// Mitsubishi GX Works2 project: Group4_V9   PLC: FX3G

// global labels: Global1
VAR_GLOBAL
  On_Switch AT X007 : BOOL;
END_VAR
VAR_GLOBAL CONSTANT
  Min_Cream : REAL := 300;
  Min_Biscuit : REAL := 6;
  Min_Choc : REAL := 120;
END_VAR
VAR_GLOBAL
  light AT Y007 : BOOL;
  Piping_Start AT X011 : BOOL;
  Whipped_Cream_Piping AT D2100 : REAL;
  Start_System AT X010 : BOOL;
  System_On AT M0 : BOOL;
  Malfunction_Status AT X005 : BOOL;
  Sen_Touch AT X001 : BOOL;
  Sen_Camera AT X002 : BOOL;
  Sen_30 AT X003 : BOOL;
  Machine AT Y004 : BOOL;
  Sen_15 AT X004 : BOOL;
  Biscuit_tray AT D2300 : REAL;
  ziluf AT M2 : BOOL;
  Blink AT M1 : BOOL;
  Blink1 AT Y000 : BOOL;
  TS_1 AT TS1 : BOOL;
  TS_2 AT TS2 : BOOL;
  Blink2 AT Y001 : BOOL;
  Check_Inv AT M17 : BOOL;
  Start_Day AT M1 : BOOL;
  Biscuit_Input AT D1333 : REAL;
  Chocolate_Input AT D1222 : REAL;
  Whipped_Cream_Input AT D1111 : REAL;
  Biscuit_Inv AT D1300 : REAL;
  Chocolate_Inv AT D1200 : REAL;
  Whipped_Cream_Inv AT D1100 : REAL;
  Full_Inv AT M107 : BOOL;
  Factory_working AT M117 : BOOL;
  Biscuit_Suff AT M130 : BOOL;
  Chocolate_Suff AT M120 : BOOL;
  Cream_Suff AT M110 : BOOL;
  Start_Glaze AT X006 : BOOL;
END_VAR
VAR_GLOBAL CONSTANT
  Double_Layer : INT := 6;
  Single_Layer : REAL := 5;
END_VAR
VAR_GLOBAL
  analog_Input_1 AT D8280 : INT;
  Single_Layer_Only AT M30 : BOOL;
END_VAR
VAR_GLOBAL CONSTANT
  Double_Layer_Amount : REAL := 240;
  Single_Layer_Amount : REAL := 120;
END_VAR
VAR_GLOBAL
  Chocolate_Dipping AT D2200 : REAL;
  Dipping_Time AT TC5 : BOOL;
  Dipping_Timer AT TC5 : BOOL;
  Dipping_Light AT Y003 : BOOL;
END_VAR
VAR_GLOBAL CONSTANT
  Double_Layer_Min : REAL := 6;
  Double_Layer_Max : REAL := 10;
  normalization : REAL := 390;
END_VAR
VAR_GLOBAL
  AnalogInput AT M33 : BOOL;
  Dip_Option AT D2220 : REAL;
  DSSD AT Y002 : BOOL;
  End_Packing AT Y002 : BOOL;
  TCoil0 AT TC0 : BOOL;
  MachineB AT D2400 : REAL;
  M_11 AT M11 : BOOL;
  TCoil1 AT TC1 : BOOL;
  M_7 AT M7 : BOOL;
  TCoil2 AT TC2 : BOOL;
  Dipping_Done AT M333 : BOOL;
  Packing_Creambo AT X000 : BOOL;
  Creambo_Counter AT CC1 : BOOL;
END_VAR
VAR_GLOBAL CONSTANT
  Creambo_5 : INT := 5;
END_VAR
VAR_GLOBAL
  Creambo_Counter_On AT CS1 : BOOL;
  last_Creambo_Warning AT Y002 : BOOL;
  Done_Packing_Counter AT CC2 : BOOL;
END_VAR
VAR_GLOBAL CONSTANT
  All_Creambo_packed : INT := 6;
END_VAR
VAR_GLOBAL
  Creambo_Done_counter AT CS2 : BOOL;
  Finished_Creambos_Sum AT D6666 : REAL;
END_VAR
VAR_GLOBAL CONSTANT
  Packed_Creambo_sixpack : REAL := 6;
END_VAR
VAR_GLOBAL
  Finished_Iteration AT M238 : BOOL;
  TC_7 AT TC7 : BOOL;
  TS_90 AT TS90 : BOOL;
  M_20 AT M20 : BOOL;
  Piping_Finished AT M200 : BOOL;
  Reset_Iteration AT M2000 : BOOL;
  Start_Glaze_Ready AT M106 : BOOL;
  Choc_Inv AT M120 : BOOL;
  Turn_Off_Inv_Check AT M227 : BOOL;
  Turn_Off_Help_Lights AT M227 : BOOL;
  TCoil3 AT TC3 : BOOL;
  TS_3 AT TS3 : BOOL;
  light_flick AT M52 : BOOL;
  TS_0 AT TS0 : BOOL;
  analog_output AT D8282 : INT;
  M_6 AT M6 : BOOL;
  M_8 AT M8 : BOOL;
END_VAR
VAR_GLOBAL CONSTANT
  normalization_back : REAL := 40;
END_VAR
VAR_GLOBAL
  M_98 AT M98 : BOOL;
  M_88 AT M88 : BOOL;
  TS_67 AT TS67 : BOOL;
  TCoil4 AT TC4 : BOOL;
  TS_4 AT TS4 : BOOL;
  M_56 AT M56 : BOOL;
  last_Iteration AT M255 : BOOL;
  Creambo_Normalized AT D6060 : REAL;
END_VAR

// task Task_01 (event TRUE, interval 0, priority 31): POU_01

PROGRAM POU_01
VAR CONSTANT
  M_10 : BOOL;
END_VAR
(* structured ladder/FBD written out as ST: instructions are called as NAME(EN, inputs, outputs); _pN, _eN, _tN stand for wires *)
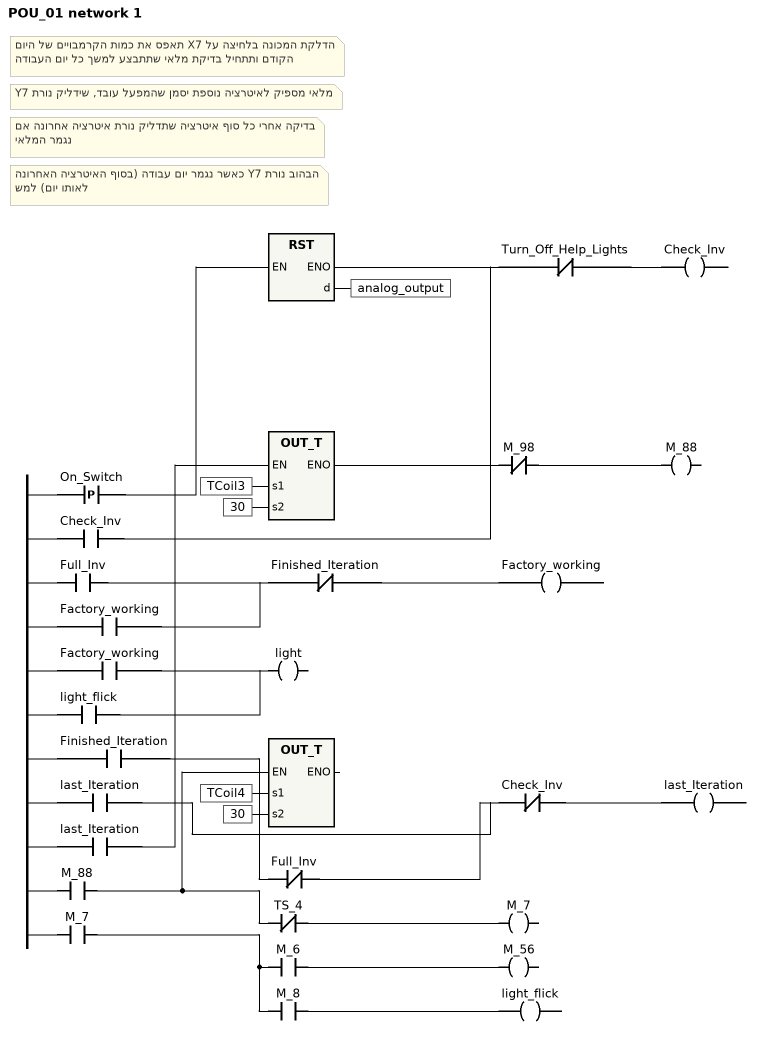
(* network 1 *)
(* הדלקת המכונה בלחיצה על X7 תאפס את כמות הקרמבויים של היום הקודם ותתחיל בדיקת מלאי שתתבצע למשך כל יום העבודה *)
(* מלאי מספיק לאיטרציה נוספת יסמן שהמפעל עובד, שידליק נורת Y7 *)
(* בדיקה אחרי כל סוף איטרציה שתדליק נורת איטרציה אחרונה אם נגמר המלאי *)
(* הבהוב נורת Y7 כאשר נגמר יום עבודה (בסוף האיטרציה האחרונה לאותו יום) למש *)
_e1 := RST(LDP(TRUE, On_Switch), analog_output);
Check_Inv := (_e1 OR Check_Inv) AND NOT Turn_Off_Help_Lights;
Factory_working := (Full_Inv OR Factory_working) AND NOT Finished_Iteration;
light := Factory_working OR light_flick;
last_Iteration := ((Finished_Iteration AND NOT Full_Inv) OR last_Iteration) AND NOT Check_Inv;
_e2 := OUT_T(last_Iteration, TCoil3, 30);
M_88 := _e2 AND NOT M_98;
OUT_T(M_88, TCoil4, 30);
M_7 := M_88 AND NOT TS_4;
M_56 := M_7 AND M_6;
light_flick := M_7 AND M_8;
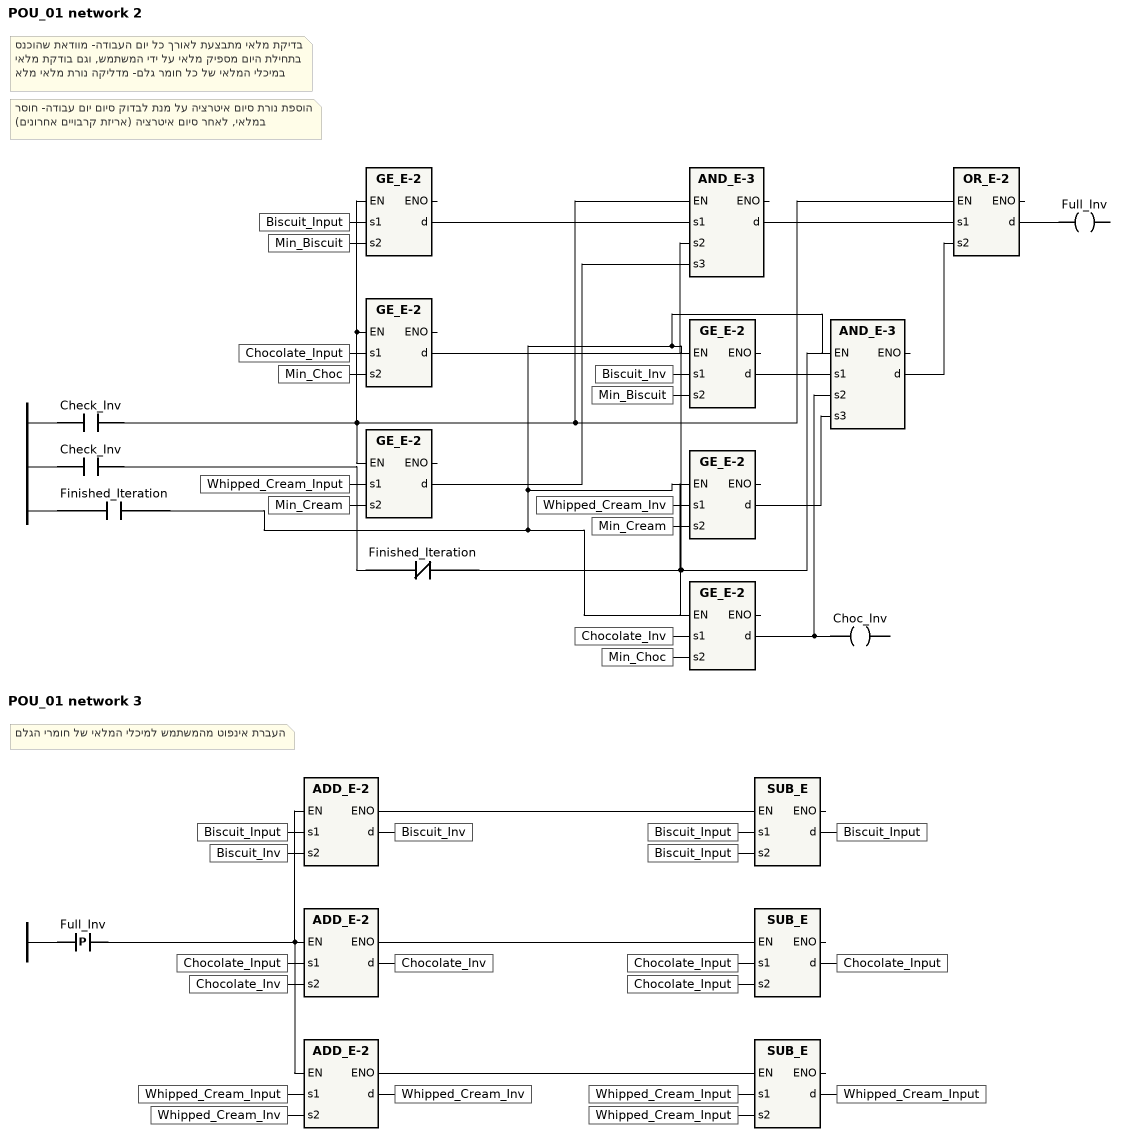
(* network 2 *)
(* בדיקת מלאי מתבצעת לאורך כל יום העבודה- מוודאת שהוכנס בתחילת היום מספיק מלאי על ידי המשתמש, וגם בודקת מלאי במיכלי המלאי של כל חומר גלם- מדליקה נורת מלאי מלא *)
(* הוספת נורת סיום איטרציה על מנת לבדוק סיום יום עבודה- חוסר במלאי, לאחר סיום איטרציה (אריזת קרבויים אחרונים) *)
GE_E(Check_Inv, Biscuit_Input, Min_Biscuit, _t1);
GE_E(Check_Inv, Chocolate_Input, Min_Choc, _t2);
GE_E(Check_Inv, Whipped_Cream_Input, Min_Cream, _t3);
AND_E(Check_Inv, _t1, _t2, _t3, _t4);
_p5 := (Check_Inv AND NOT Finished_Iteration) OR Finished_Iteration;
GE_E(_p5, Biscuit_Inv, Min_Biscuit, _t6);
GE_E(_p5, Chocolate_Inv, Min_Choc, _t7);
GE_E(_p5, Whipped_Cream_Inv, Min_Cream, _t8);
AND_E(_p5, _t6, _t7, _t8, _t9);
OR_E(Check_Inv, _t4, _t9, _t10);
Full_Inv := _t10;
Choc_Inv := _t7;
(* network 3 *)
(* העברת אינפוט מהמשתמש למיכלי המלאי של חומרי הגלם *)
_p1 := LDP(TRUE, Full_Inv);
_e2 := ADD_E(_p1, Biscuit_Input, Biscuit_Inv, Biscuit_Inv);
SUB_E(_e2, Biscuit_Input, Biscuit_Input, Biscuit_Input);
_e3 := ADD_E(_p1, Chocolate_Input, Chocolate_Inv, Chocolate_Inv);
SUB_E(_e3, Chocolate_Input, Chocolate_Input, Chocolate_Input);
_e4 := ADD_E(_p1, Whipped_Cream_Input, Whipped_Cream_Inv, Whipped_Cream_Inv);
SUB_E(_e4, Whipped_Cream_Input, Whipped_Cream_Input, Whipped_Cream_Input);
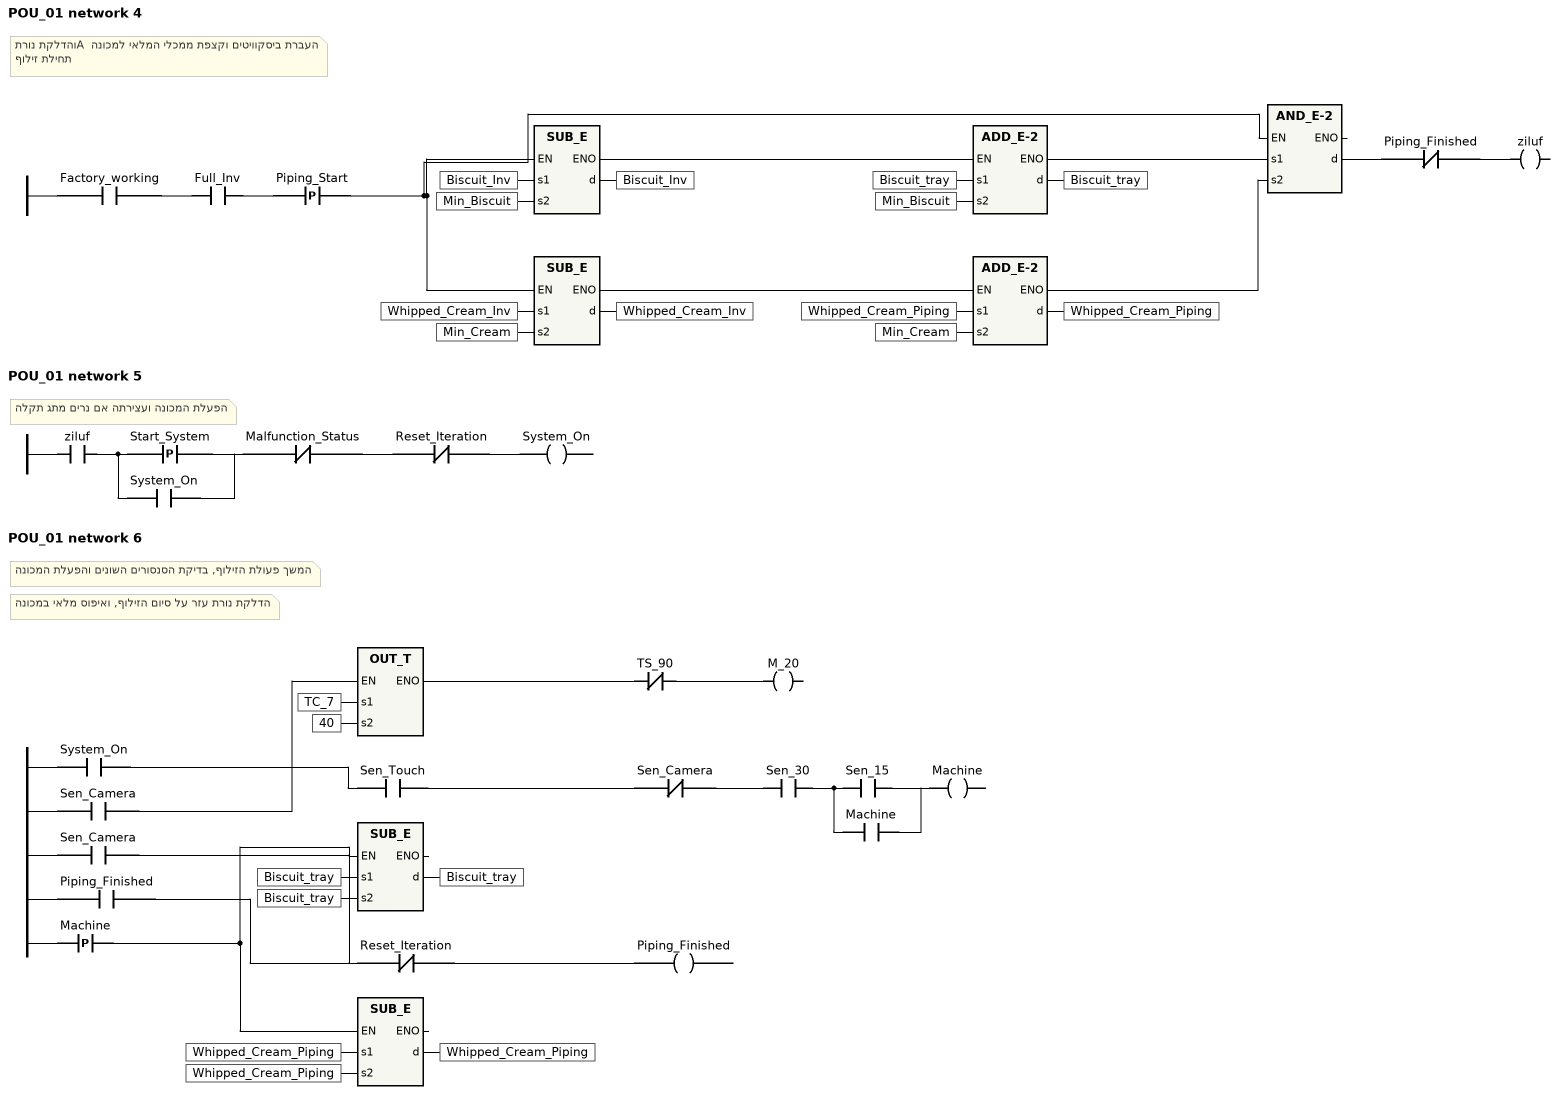
(* network 4 *)
(* העברת ביסקוויטים וקצפת ממכלי המלאי למכונה  Aוהדלקת נורת תחילת זילוף *)
_p1 := Factory_working AND Full_Inv AND LDP(TRUE, Piping_Start);
_e2 := SUB_E(_p1, Biscuit_Inv, Min_Biscuit, Biscuit_Inv);
_e3 := ADD_E(_e2, Biscuit_tray, Min_Biscuit, Biscuit_tray);
_e4 := SUB_E(_p1, Whipped_Cream_Inv, Min_Cream, Whipped_Cream_Inv);
_e5 := ADD_E(_e4, Whipped_Cream_Piping, Min_Cream, Whipped_Cream_Piping);
AND_E(_p1, _e3, _e5, _t6);
ziluf := _t6 AND NOT Piping_Finished;
(* network 5 *)
(* הפעלת המכונה ועצירתה אם נרים מתג תקלה *)
System_On := (((ziluf AND LDP(TRUE, Start_System)) OR (ziluf AND System_On)) AND NOT Malfunction_Status) AND NOT Reset_Iteration;
(* network 6 *)
(* המשך פעולת הזילוף, בדיקת הסנסורים השונים והפעלת המכונה *)
(* הדלקת נורת עזר על סיום הזילוף, ואיפוס מלאי במכונה *)
_p1 := System_On AND Sen_Touch AND NOT Sen_Camera AND Sen_30;
Machine := (_p1 AND Sen_15) OR (_p1 AND Machine);
_e2 := OUT_T(Sen_Camera, TC_7, 40);
M_20 := _e2 AND NOT TS_90;
Piping_Finished := (Sen_Camera OR Piping_Finished) AND NOT Reset_Iteration;
_p3 := LDP(TRUE, Machine);
SUB_E(_p3, Biscuit_tray, Biscuit_tray, Biscuit_tray);
SUB_E(_p3, Whipped_Cream_Piping, Whipped_Cream_Piping, Whipped_Cream_Piping);
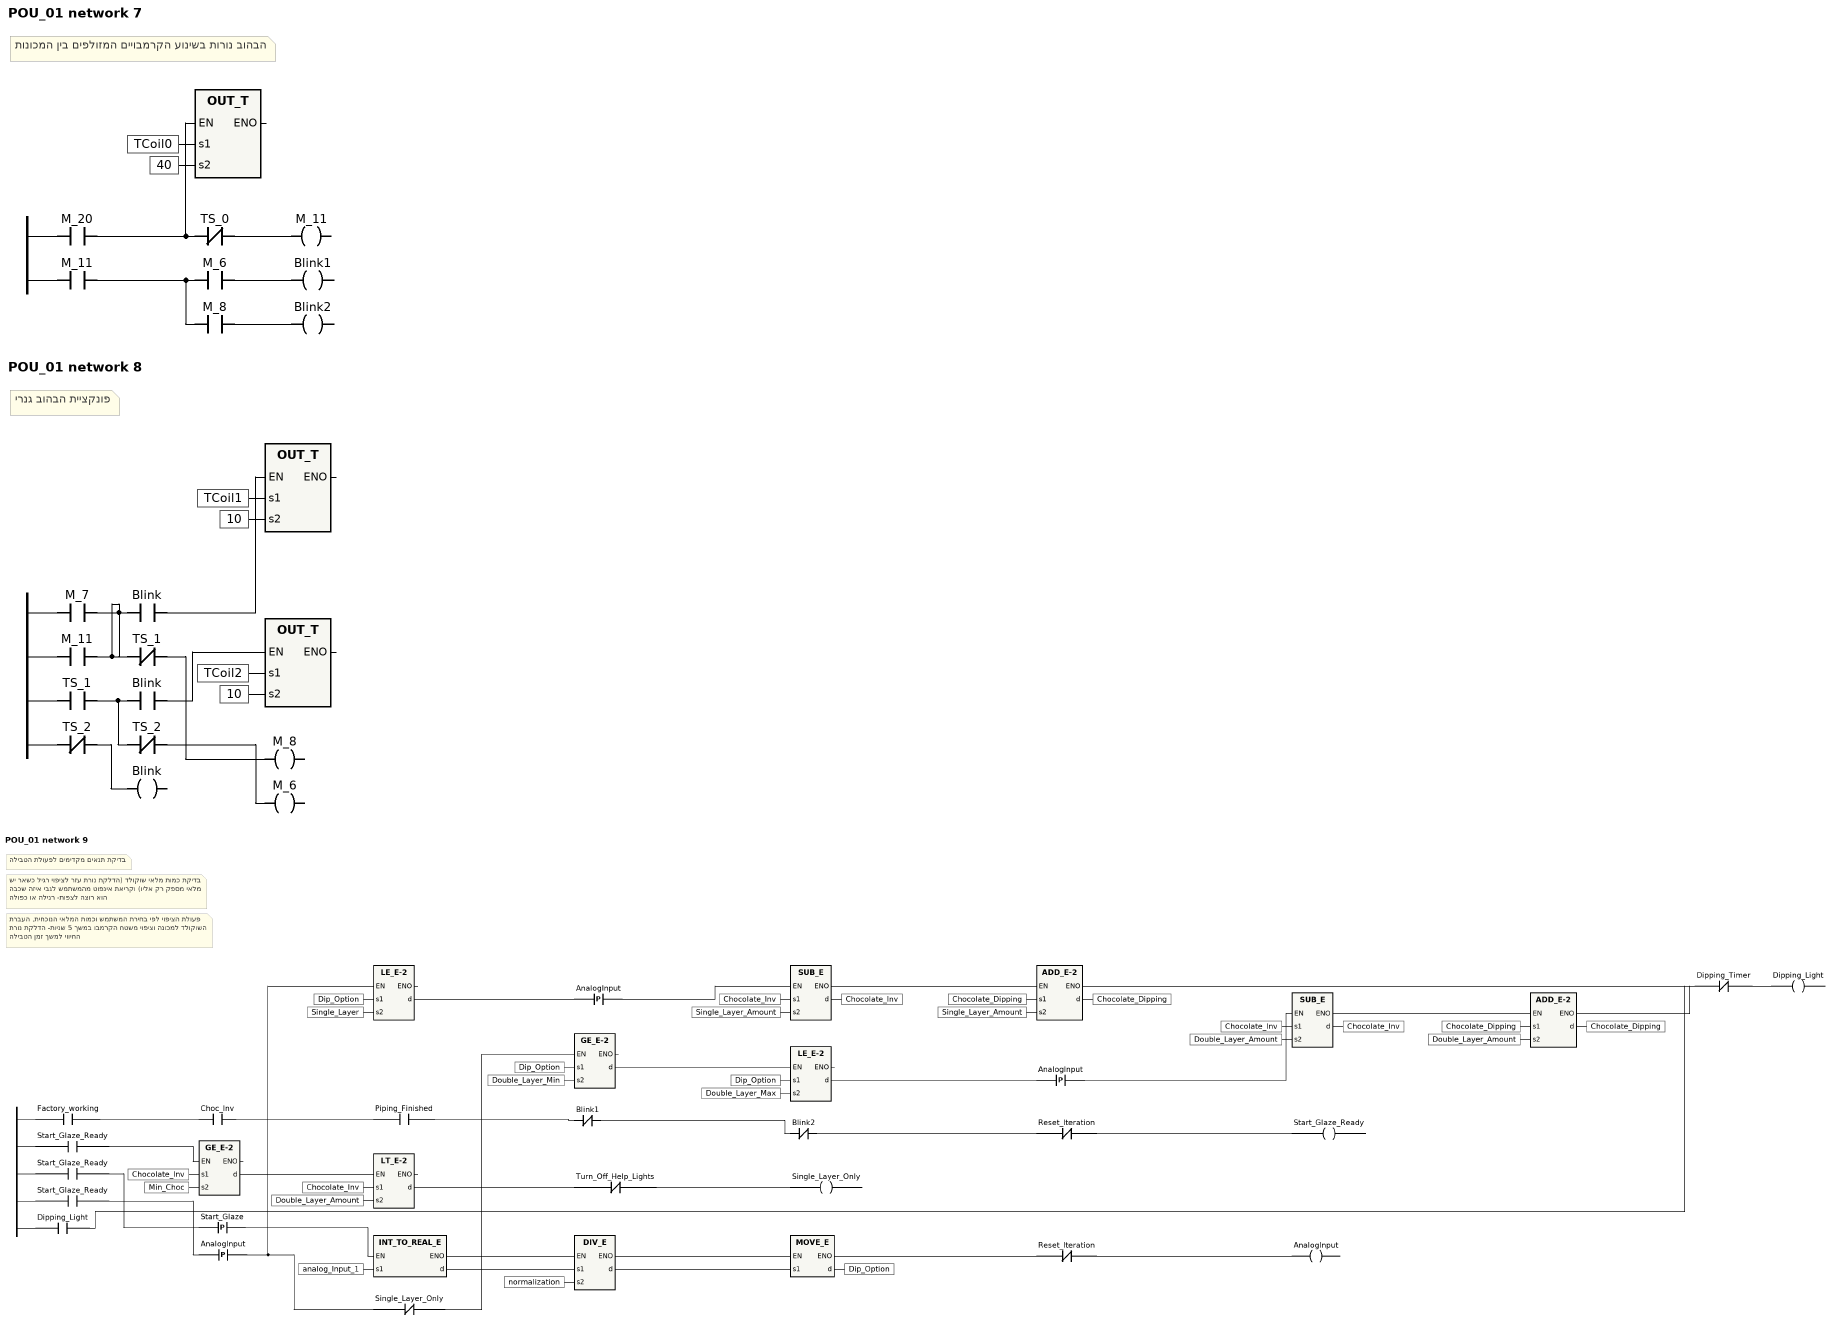
(* network 7 *)
(* הבהוב נורות בשינוע הקרמבויים המזולפים בין המכונות *)
OUT_T(M_20, TCoil0, 40);
M_11 := M_20 AND NOT TS_0;
Blink1 := M_11 AND M_6;
Blink2 := M_11 AND M_8;
(* network 8 *)
(* פונקציית הבהוב גנרי *)
_p1 := M_7 OR M_11;
OUT_T(_p1 AND Blink, TCoil1, 10);
M_8 := _p1 AND NOT TS_1;
OUT_T(TS_1 AND Blink, TCoil2, 10);
M_6 := TS_1 AND NOT TS_2;
Blink := NOT TS_2;
(* network 9 *)
(* בדיקת תנאים מקדימים לפעולת הטבילה *)
(* בדיקת כמות מלאי שוקולד (הדלקת נורת עזר לציפוי רגיל כשאר יש מלאי מספק רק אליו) וקריאת אינפוט מהמשתמש לגבי איזה שכבה הוא רוצה לצפות- רגילה או כפולה *)
(* פעולת הציפוי לפי בחירת המשתמש וכמות המלאי הנוכחית, העברת השוקולד למכונה וציפוי משטח הקרמבו במשך 5 שניות- הדלקת נורת החיווי למשך זמן הטבילה *)
Start_Glaze_Ready := Factory_working AND Choc_Inv AND Piping_Finished AND NOT Blink1 AND NOT Blink2 AND NOT Reset_Iteration;
GE_E(Start_Glaze_Ready, Chocolate_Inv, Min_Choc, _t1);
LT_E(_t1, Chocolate_Inv, Double_Layer_Amount, _t2);
Single_Layer_Only := _t2 AND NOT Turn_Off_Help_Lights;
_e4 := INT_TO_REAL_E(Start_Glaze_Ready AND LDP(TRUE, Start_Glaze), analog_Input_1, _t3);
_e6 := DIV_E(_e4, _t3, normalization, _t5);
_e7 := MOVE_E(_e6, _t5, Dip_Option);
AnalogInput := _e7 AND NOT Reset_Iteration;
_p8 := Start_Glaze_Ready AND LDP(TRUE, AnalogInput);
LE_E(_p8, Dip_Option, Single_Layer, _t9);
_e10 := SUB_E(_t9 AND LDP(TRUE, AnalogInput), Chocolate_Inv, Single_Layer_Amount, Chocolate_Inv);
_e11 := ADD_E(_e10, Chocolate_Dipping, Single_Layer_Amount, Chocolate_Dipping);
GE_E(_p8 AND NOT Single_Layer_Only, Dip_Option, Double_Layer_Min, _t12);
LE_E(_t12, Dip_Option, Double_Layer_Max, _t13);
_e14 := SUB_E(_t13 AND LDP(TRUE, AnalogInput), Chocolate_Inv, Double_Layer_Amount, Chocolate_Inv);
_e15 := ADD_E(_e14, Chocolate_Dipping, Double_Layer_Amount, Chocolate_Dipping);
Dipping_Light := (_e11 OR _e15 OR Dipping_Light) AND NOT Dipping_Timer;
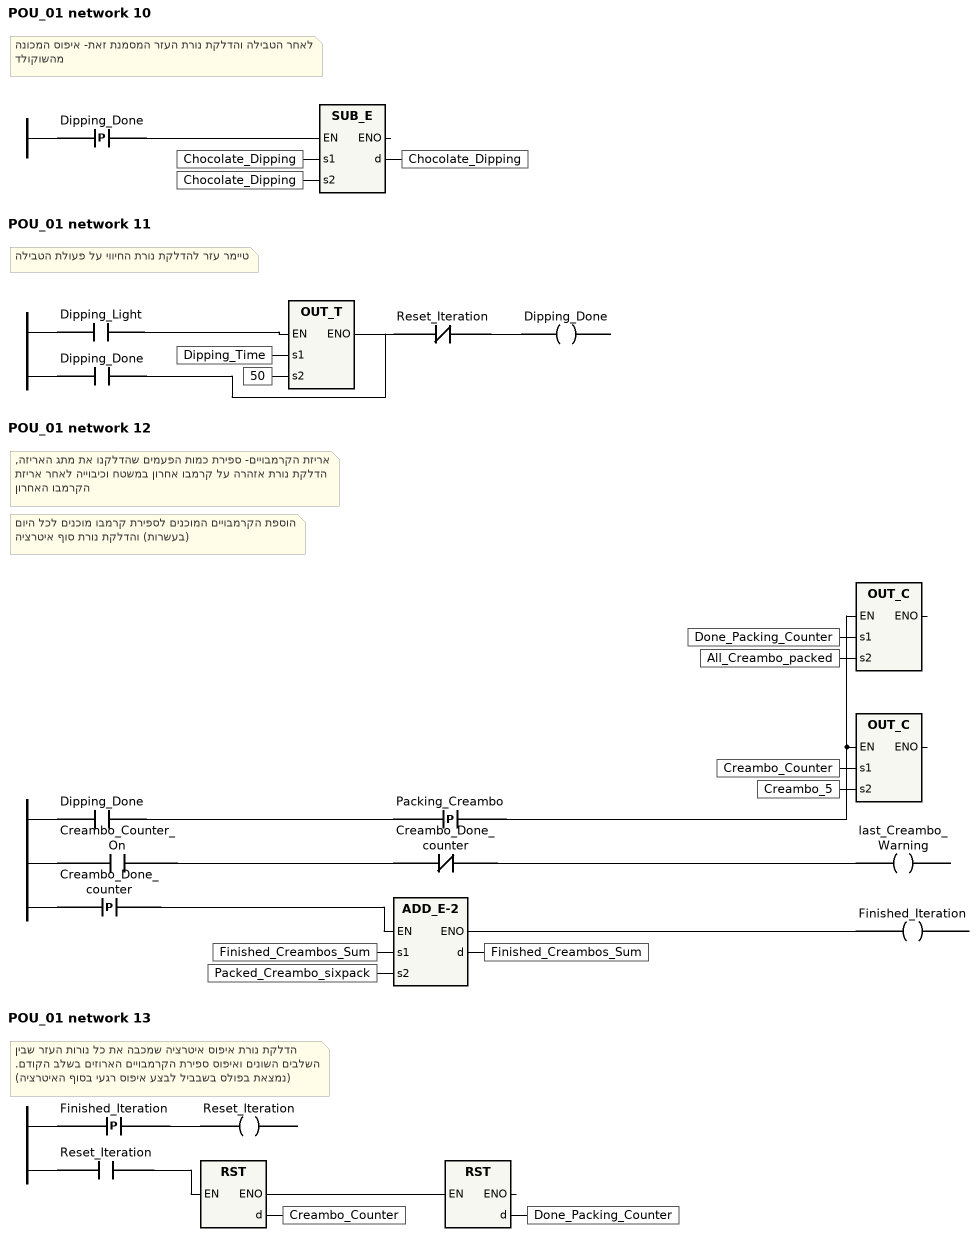
(* network 10 *)
(* לאחר הטבילה והדלקת נורת העזר המסמנת זאת- איפוס המכונה מהשוקולד *)
SUB_E(LDP(TRUE, Dipping_Done), Chocolate_Dipping, Chocolate_Dipping, Chocolate_Dipping);
(* network 11 *)
(* טיימר עזר להדלקת נורת החיווי על פעולת הטבילה *)
_e1 := OUT_T(Dipping_Light, Dipping_Time, 50);
Dipping_Done := (_e1 OR Dipping_Done) AND NOT Reset_Iteration;
(* network 12 *)
(* אריזת הקרמבויים- ספירת כמות הפעמים שהדלקנו את מתג האריזה, הדלקת נורת אזהרה על קרמבו אחרון במשטח וכיבוייה לאחר אריזת הקרמבו האחרון *)
(* הוספת הקרמבויים המוכנים לספירת קרמבו מוכנים לכל היום (בעשרות) והדלקת נורת סוף איטרציה *)
_p1 := Dipping_Done AND LDP(TRUE, Packing_Creambo);
OUT_C(_p1, Done_Packing_Counter, All_Creambo_packed);
OUT_C(_p1, Creambo_Counter, Creambo_5);
last_Creambo_Warning := Creambo_Counter_On AND NOT Creambo_Done_counter;
_e2 := ADD_E(LDP(TRUE, Creambo_Done_counter), Finished_Creambos_Sum, Packed_Creambo_sixpack, Finished_Creambos_Sum);
Finished_Iteration := _e2;
(* network 13 *)
(* הדלקת נורת איפוס איטרציה שמכבה את כל נורות העזר שבין השלבים השונים ואיפוס ספירת הקרמבויים הארוזים בשלב הקודם. (נמצאת בפולס בשבביל לבצע איפוס רגעי בסוף האיטרציה) *)
Reset_Iteration := LDP(TRUE, Finished_Iteration);
_e1 := RST(Reset_Iteration, Creambo_Counter);
RST(_e1, Done_Packing_Counter);
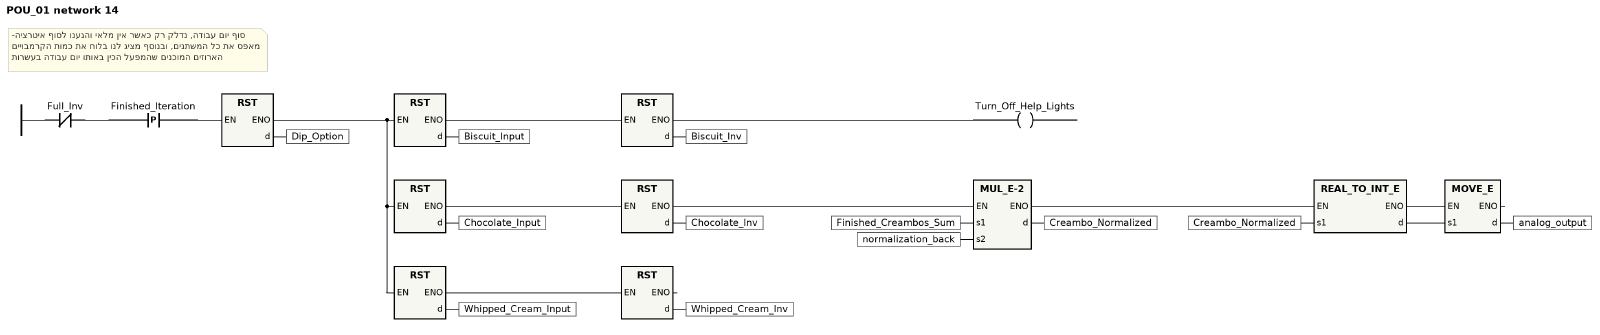
(* network 14 *)
(* סוף יום עבודה, נדלק רק כאשר אין מלאי והגענו לסוף איטרציה- מאפס את כל המשתנים, ובנוסף מציג לנו בלוח את כמות הקרמבויים הארוזים המוכנים שהמפעל הכין באותו יום עבודה בעשרות *)
_e1 := RST(NOT Full_Inv AND LDP(TRUE, Finished_Iteration), Dip_Option);
_e2 := RST(_e1, Biscuit_Input);
_e3 := RST(_e2, Biscuit_Inv);
Turn_Off_Help_Lights := _e3;
_e4 := RST(_e1, Chocolate_Input);
_e5 := RST(_e4, Chocolate_Inv);
_e6 := MUL_E(_e5, Finished_Creambos_Sum, normalization_back, Creambo_Normalized);
_e8 := REAL_TO_INT_E(_e6, Creambo_Normalized, _t7);
MOVE_E(_e8, _t7, analog_output);
_e9 := RST(_e1, Whipped_Cream_Input);
RST(_e9, Whipped_Cream_Inv);
END_PROGRAM
